GLOBALCONSTANTS Global_NAME_Functions (* Industry non-specific function defines *)
  (* Standard: 61499-1 *)
  (* Version 1.0, 2026-06-29, Franz Höpfinger, Demmler Andreas Fahrzeugbau *)
  PACKAGE isobus::pgn::const;
  VAR_GLOBAL CONSTANT
    F_ENGINE : BYTE := 0; (* Function: Engine - While the function identifies what is typically the mechanical power source of *)
    F_AUX_POWER_UNIT : BYTE := 1; (* Function: Auxiliary Power Unit (APU) - Power source for operating systems without the use of the *)
    F_ELEC_PROPULSION_CONTROL : BYTE := 2; (* Function: Electric Propulsion Control - Control system which operates the drive mechanism when it *)
    F_TRANSMISSION : BYTE := 3; (* Function: Transmission - A mechanical system for alter the speed vs torque output of the engine *)
    F_BATTERY_PACK_MONITOR : BYTE := 4; (* Function: Battery Pack Monitor - Monitors the condition - charge, temperature, power remaining, *)
    F_SHIFT_CONTROL_CONSOLE : BYTE := 5; (* Function: Shift Control/Console - The device which determines and transmit onto the network the *)
    F_POWER_TAKEOFF_MAIN_OR_REAR : BYTE := 6; (* Function: Power TakeOff - (Main or Rear) - The system which controls the mechanical power derived *)
    F_AXLE_STEERING : BYTE := 7; (* Function: Axle - Steering - Adjust attack angle as function of steering *)
    F_AXLE_DRIVE : BYTE := 8; (* Function: Axle - Drive *)
    F_BRAKES_SYSTEMCONTROL : BYTE := 9; (* Function: Brakes - System Controller - Controls service braking system electronically – might be *)
    F_BRAKES_STEER_AXLE : BYTE := 10; (* Function: Brakes - Steer Axle - Control for actuating the service brakes on a steered axle *)
    F_BRAKES_DRIVE_AXLE : BYTE := 11; (* Function: Brakes - Drive axle - Control for actuating the service brakes on a drive axle *)
    F_RETARDER_ENGINE : BYTE := 12; (* Function: Retarder - Engine - The control for the retarder capabilities of the engine. There are *)
    F_RETARDER_DRIVELINE : BYTE := 13; (* Function: Retarder - Driveline - The control for the retarder capabilities of the driveline. *)
    F_CRUISE_CONTROL : BYTE := 14; (* Function: Cruise Control - Control system for maintaining the vehicle’s speed at a fixed operator *)
    F_FUEL_SYSTEM : BYTE := 15; (* Function: Fuel System - Controls fuel flow from the tank to the filter to the *)
    F_STEERING_CONTROL : BYTE := 16; (* Function: Steering Controller - Controls steering in steer-by-wire *)
    F_SUSPENSION_STEER_AXLE : BYTE := 17; (* Function: Suspension - Steer Axle - Control system for the suspension of a steered axle *)
    F_SUSPENSION_DRIVE_AXLE : BYTE := 18; (* Function: Suspension - Drive Axle - Control system for the suspension of a driven axle *)
    F_INSTRUMENT_CLUSTER : BYTE := 19; (* Function: Instrument Cluster - A gauge display for a vehicle. Typically mounted in the cab within *)
    F_TRIP_RECORDER : BYTE := 20; (* Function: Trip Recorder - A system for accumulating data versus travel of the vehicle (machine), *)
    F_CAB_CLIMATE_CONTROL : BYTE := 21; (* Function: Cab Climate Control - A system for controlling the climate within the cab of the *)
    F_AERODYNAMIC_CONTROL : BYTE := 22; (* Function: Aerodynamic Control - Modify drag by altering Body panels – lower air ferrings when *)
    F_VEHICLE_NAVIGATION : BYTE := 23; (* Function: Vehicle Navigation - System associated with the vehicles physical location – may be as *)
    F_VEHICLE_SECURITY : BYTE := 24; (* Function: Vehicle Security - System for comparing operator provided data sequences against *)
    F_NETWORK_INTERCONNECT_UNIT : BYTE := 25; (* Function: Network Interconnect ECU - ECU for connecting different network segments together – may *)
    F_BODY_CONTROLLER : BYTE := 26; (* Function: Body Controller - May handle suspension control for the body sections independent from *)
    F_POWER_TAKEOFF_SECONDARY_OR_FRONT : BYTE := 27; (* Function: Power TakeOff (Secondary or Front) - The system which controls the mechanical power *)
    F_OFF_VEHICLE_GATEWAY : BYTE := 28; (* Function: Off Vehicle Gateway - ECU for connecting between vehicle network(s) and an off-vehicle *)
    F_VTERMINAL : BYTE := 29; (* Function: Virtual Terminal (in cab) - A general purpose ‘intelligent’ display with a specific *)
    F_MANAGEMENT_COMPUTER : BYTE := 30; (* Function: Management Computer - Manages vehicle systems, i.e. powertrain. *)
    F_PROPULSION_BATTERY_CHARGER : BYTE := 31; (* Function: Propulsion Battery Charger - A device used to charge propulsion batteries in an *)
    F_HEADWAY_CONTROLLER : BYTE := 32; (* Function: Headway Controller - Forward-looking collision avoidance, collision warning, speed *)
    F_SYSTEM_MONITOR : BYTE := 33; (* Function: System Monitor *)
    F_HYDRAULIC_PUMP_CONTROLLER : BYTE := 34; (* Function: Hydraulic Pump Controller - Pump which provides hydraulic power to operate installed *)
    F_SUSPENSION_SYSTEM_CONTROLLER : BYTE := 35; (* Function: Suspension - System Controller - A controller responsible for co-ordinating the *)
    F_PNEUMATIC_SYSTEM_CONTROLLER : BYTE := 36; (* Function: Pneumatic - System Controller *)
    F_CAB_CONTROLLER : BYTE := 37; (* Function: Cab Controller - A controller located in/near vehicle cab to perform functions that are *)
    F_TIRE_PRESSURE_CONTROL : BYTE := 38; (* Function: Tire Pressure Control - The device providing centralised tire inflation *)
    F_IGNITION_CONTROL_MODULE : BYTE := 39; (* Function: Ignition Control Module - A device for altering the ignition of an engine and with *)
    F_SEAT_CONTROL : BYTE := 40; (* Function: Seat Control - A system for controlling the seats (operator and passenger) within the *)
    F_LIGHTING_OPERATOR_CONTROLS : BYTE := 41; (* Function: Lighting - Operator Controls - The controller for sending the operator lighting *)
    F_WATER_PUMP_CONTROL : BYTE := 42; (* Function: Water Pump Control - Controller for a water pump mounted on the vehicle/machine. For *)
    F_TRANSMISSION_DISPLAY : BYTE := 43; (* Function: Transmission Display - Display designed specifically to display transmission *)
    F_EXHAUST_EMISSION_CONTROL : BYTE := 44; (* Function: Exhaust Emission Control *)
    F_VEHICLE_DYNAMIC_STABILITY_CONTROL : BYTE := 45; (* Function: Vehicle Dynamic Stability Control *)
    F_OIL_SENSOR_UNIT : BYTE := 46; (* Function: Oil Sensor Unit *)
    F_INFORMATION_SYSTEM_CONTROLLER : BYTE := 47; (* Function: Information System Controller - Information management for the vehicle's application, *)
    F_RAMP_CONTROL : BYTE := 48; (* Function: Ramp Control - Loading unloading – chairlift, ramps, lifts, or tailgates *)
    F_CLUTCH_CONVERTER_CONTROL : BYTE := 49; (* Function: Clutch/Converter Control - When transmission is distributed this handles torque *)
    F_AUXILIARY_HEATER : BYTE := 50; (* Function: Auxiliary Heater - Primary heat is typically taken from the engine coolant. This is the *)
    F_FORWARD_LOOKING_COLLISION_WARNING_SYSTEM : BYTE := 51; (* Function: Forward-Looking Collision Warning System - A system which detects and warns of *)
    F_CHASSIS_CONTROLLER : BYTE := 52; (* Function: Chassis Controller - Controls the chassis (not body or cab) components *)
    F_ALTERNATOR_CHARGING_SYSTEM : BYTE := 53; (* Function: Alternator/Charging System - Vehicle's primary on-board charging controller - *)
    F_COMMUNICATIONS_UNIT_CELLULAR : BYTE := 54; (* Function: Communications Unit, Cellular - Radio communications device designed specifically to *)
    F_COMMUNICATIONS_UNIT_SATELLITE : BYTE := 55; (* Function: Communications Unit, Satellite - Radio communications device designed specifically to *)
    F_COMMUNICATIONS_UNIT_RADIO : BYTE := 56; (* Function: Communications Unit, Radio - Radio communications device designed specifically to *)
    F_AUXILIARY_DEVICE : BYTE := 57; (* Function: Steering Column Unit - Device that gathers the operator inputs from switches/levers/etc *)
    F_FAN_DRIVE_CONTROL : BYTE := 58; (* Function: Fan Drive Control - Primary control system affecting the operation of the main cooling *)
    F_STARTER : BYTE := 59; (* Function: Starter - A mechanical system for initiating rotation in an engine that is stopped. *)
    F_CAB_DISPLAY : BYTE := 60; (* Function: Cab Display - Cab Display is for a fairly elaborate in cab display, typically capable *)
    F_FILESERVER : BYTE := 61; (* Function: File Server / Printer - A printing or file storage unit on the network - A permanent *)
    F_ON_BOARD_DIAGNOSTIC_UNIT : BYTE := 62; (* Function: On-Board Diagnostic Unit - A tool which may be permanently mounted on the vehicle and *)
    F_ENGINE_VALVE_CONTROLLER : BYTE := 63; (* Function: Engine Valve Controller - Control system used to manipulate the actuation of engine *)
    F_ENDURANCE_BRAKING : BYTE := 64; (* Function: Endurance Braking - Sum of all devices in a vehicle which enable the driver with *)
    F_GAS_FLOW_MEASUREMENT : BYTE := 65; (* Function: Gas Flow Measurement - Provides measurement of gas flow rates and associated *)
    F_I_O_CONTROLLER : BYTE := 66; (* Function: I/O Controller - Reporting and/or control device for external input and output channels *)
    F_ELECTRICAL_SYSTEM_CONTROLLER : BYTE := 67; (* Function: Electrical System Controller - This may include Load Centers, Fuseboxes, & Power *)
    F_AFTERTREATMENT_SYSTEM_GAS_MEASUREMENT : BYTE := 68; (* Function: Aftertreatment system gas measurement - Sensor for measuring gas properties before and *)
    F_ENGINE_EMISSION_AFTERTREATMENT_SYSTEM : BYTE := 69; (* Function: Engine Emission Aftertreatment System - Engine Emission Aftertreatment System *)
    F_AUXILIARY_REGENERATION_DEVICE : BYTE := 70; (* Function: Auxiliary Regeneration Device - Auxiliary Regeneration Device used as part of an after *)
    F_TRANSFER_CASE_CONTROL : BYTE := 71; (* Function: Transfer Case Control - The device which controls the selection of the number of drive *)
    F_COOLANT_VALVE_CONTROLLER : BYTE := 72; (* Function: Coolant Valve Controller - Device used to control the flow of coolant (water, oil, air, *)
    F_ROLLOVER_DETECTION_CONTROL : BYTE := 73; (* Function: Rollover Detection Control - Device designed for detection of vehicle rollover. *)
    F_LUBRICATION_SYSTEM : BYTE := 74; (* Function: Lubrication System - The Lubrication System pumps quantities of lubricant to each *)
    F_SUPPLEMENTAL_FAN : BYTE := 75; (* Function: Supplemental Fan - This is an auxillary fan used for additional cooling. It is in *)
    F_TEMPERATURE_SENSOR : BYTE := 76; (* Function: Temperature Sensor - Device which measures temperature. *)
    F_FUEL_PROPERTIES_SENSOR : BYTE := 77; (* Function: Fuel Properties Sensor - Device which measures fuel properties *)
    F_FIRE_SUPPRESSION_SYSTEM : BYTE := 78; (* Function: Fire Suppression System - Fire Suppression System *)
    F_POWER_SYSTEMS_MANAGER : BYTE := 79; (* Function: Power Systems Manager - Controller application that manages the power output of one or *)
    F_ELECTRIC_POWERTRAIN : BYTE := 80; (* Function: Electric Powertrain - Controller application in charge of controlling and coordinating *)
    F_HYDRAULIC_POWERTRAIN : BYTE := 81; (* Function: Hydraulic Powertrain - Controller application in charge of controlling and coordinating *)
    F_FILE_SERVER : BYTE := 82; (* Function: File Server - A file storage unit on the network - A permanent connection may exist and *)
    F_PRINTER : BYTE := 83; (* Function: Printer - A printing unit on the network - A permanent connection may exist and the *)
    F_START_AID_DEVICE : BYTE := 84; (* Function: Start Aid Device - Device that controls hardware and/or conveys information related to *)
    F_ENGINE_INJECTION_CONTROL_MODULE : BYTE := 85; (* Function: Engine Injection Control Module - A device for direct or port injection of fuel for *)
    F_EV_COMMUNICATION_CONTROLLER : BYTE := 86; (* Function: EV Communication Controller - A controller or application that manages the connection *)
    F_DRIVER_IMPAIRMENT_DEVICE : BYTE := 87; (* Function: Driver Impairment Device - Device which prevents the starting of a vehicle motor due to *)
    F_ELECTRIC_POWER_CONVERTER : BYTE := 88; (* Function: Electric Power Converter - An inverter or converter used to transform AC or DC power to *)
    F_SUPPLY_EQUIPMENT_COMMUNICATION_CONTROLLER_SECC : BYTE := 89; (* Function: Supply Equipment Communication Controller (SECC) - Typically part of an Electrical *)
    F_VEHICLE_ADAPTER_COMMUNICATION_CONTROLLER_VACC : BYTE := 90; (* Function: Vehicle Adapter Communication Controller (VACC) - A controller inside of the adapter *)
    F_ACCESSORY_ELECTRIC_MOTOR_CONTROLLER : BYTE := 91; (* Function: Accessory Electric Motor Controller - Controller responsible for the operation and *)
    F_CURRENT_SENSOR : BYTE := 92; (* Function: Current Sensor - Sensor for measuring current *)
    F_FUEL_CELL_SYSTEM : BYTE := 93; (* Function: Fuel Cell System - Controller for a system that converts fuel (e.g., hydrogen) to *)
    F_AUXILIARY_DISPLAY : BYTE := 94; (* Function: Auxiliary Display - Auxiliary Display for displaying information. It is located inside *)
    F_NOT_AVAILABLE : BYTE := 255; (* Function: not available function; used as a placeholder for all functions *)
  END_VAR
END_GLOBALCONSTANTS
